TYPE ST_MachineControl :
STRUCT
	bAuto					:BOOL;
	bManual					:BOOL;
	bMaintenance			:BOOL;
	bStart					:BOOL;
	bStop					:BOOL;
	bPause					:BOOL;
	bDoorClose				:BOOL;	
	bDoorOpen				:BOOL;
	bNext					:BOOL;
	bPrevious				:BOOL;
END_STRUCT
END_TYPE

(* stored: Version 1.1.0.1, ProductVersion 3.1.4024.12
   DUT ST_MachineControl: Id {6e52120e-a7f6-4368-af04-8e9b4da5919e} *)
